Yaskawa INFORM job: R1-R2-S1-2.JBI

/JOB
//NAME R1-R2-S1-2
//POS
///NPOS 8,0,4,0,0,0
///TOOL 0
///POSTYPE PULSE
///PULSE
C00000=-6744,-46438,-34826,-14046,-21223,6588
///TOOL 1
C00001=-6022,-65326,-52845,3,-2902,-16
///TOOL 0
C00002=-23628,-46438,-34826,-14046,-21223,6588
///TOOL 1
C00003=-26042,-65326,-52845,3,-2902,-16
///TOOL 0
C00004=-23628,-2565,-34826,-14046,-21223,6588
///TOOL 1
C00005=18046,-65326,-52845,3,-26155,-16
///TOOL 0
C00006=-42829,-2565,-34826,-14046,-21223,6588
///TOOL 1
C00007=18046,-39405,-52845,3,-26155,-16
///TOOL 0
EC00000=-28898,221232
EC00001=10741,151008
EC00002=10741,151008
EC00003=10741,151008
//INST
///DATE 2023/02/06 16:30
///ATTR SC,RW
///GROUP1 RB1,ST1
///GROUP2 RB2
NOP
MOVJ C00000 EC00000 VJ=10.00  +MOVJ C00001 VJ=10.00
MOVJ C00002 EC00001 VJ=10.00  +MOVJ C00003 VJ=10.00
MOVL C00004 EC00002 V=11.0  +MOVL C00005 V=11.0
MOVL C00006 EC00003 V=11.0  +MOVL C00007 V=11.0
END
